(* PLC project Senza_nome, Sconosciuto Senza_nome 1 *)
(* stored: creationDateTime 2026-08-25T11:15:53, modificationDateTime 2026-08-25T11:29:17 *)

PROGRAM program0
  VAR
    CTU0 : CTU;
    CU : BOOL;
    PULSE : BOOL;
    Q : BOOL;
    Reset : BOOL;
    Preset_value : INT := 5;
  END_VAR
  VAR  (* added by the conversion: wires and edge detectors of the diagram *)
    R_TRIG1 : R_TRIG;
  END_VAR

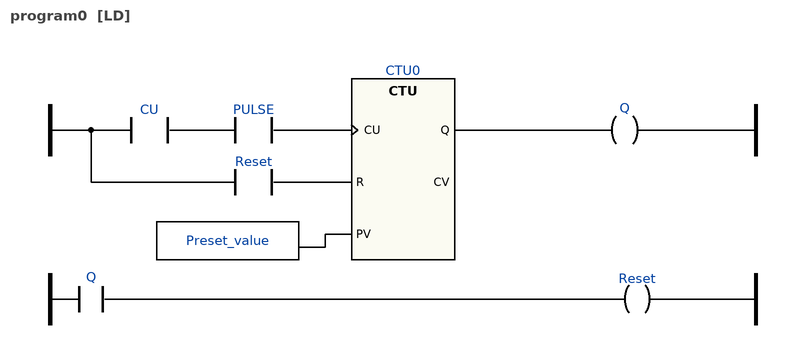
(* LD diagram, written out as Structured Text *)
R_TRIG1(CLK := CU AND PULSE);
CTU0(CU := R_TRIG1.Q, R := Reset, PV := Preset_value);
Q := CTU0.Q;
Reset := Q;
END_PROGRAM

CONFIGURATION Config0
  RESOURCE Res0 ON PLC
    TASK task0(INTERVAL := T#20ms, PRIORITY := 0);
    PROGRAM instance0 WITH task0 : program0;
  END_RESOURCE
END_CONFIGURATION
